TYPE ST_HMI_Monitor_Limits :
STRUCT
	//LIMITS
	//r_Pmin						: REAL ;
	//r_Pmax						: REAL ;
	//r_QMin						: REAL ;
	//r_QMax						: REAL ;
	r_ACcurrentLimit			: REAL;
	r_ApparentPowerlimit		: REAL;
	r_ActivePowerlimit			: REAL;
	r_DCcurrentLimit			: REAL;
	r_DroopLimit				: REAL;
	
END_STRUCT
END_TYPE

(* stored: Version 1.1.0.1, ProductVersion 3.1.4026.18
   DUT ST_HMI_Monitor_Limits: Id {7e172b71-05a7-424f-8445-5c443887ed5f} *)
